Staubli VAL3: saveOldframe.pgx

program saveOldframe()
begin
  lib:fr1.trsf=f1.trsf
  lib:t1.trsf=t1.trsf
end
